Fanuc KAREL source: NC0061.KL

-- PROVISIONAL review KL for V940-1; original PC SHA256 46cbbacf586b5ee398f1359ac13f002e54e1b3793ebfd17aa1c9afa5b6356ba0
-- Incomplete behavior may be omitted. Consult companion uncertainty JSON. Do not deploy.
PROGRAM NC0061
%NOLOCKGROUP
-- UNRESOLVED_LOCAL_POOL 1 cells at code offset 3; source declarations unknown
-- DIRECT_LOCAL_WORD_ACCESS alone does not prove INTEGER, REAL, or BOOLEAN
BEGIN
  -- V9_CONDITION_STACK_HINT 10 bounded expression windows; static native code-base-relative target link; source arms held
  -- UNRESOLVED_PC offsets 0-8; opcodes 2B,2C,7B
  -- UNRESOLVED_PC offsets 13-20; opcodes 9D,23
  -- UNRESOLVED_PC offsets 25-42; opcodes 21,40,41,42
  -- UNRESOLVED_PC offsets 47-81; opcodes 21,2E,52,23,7A,40,41,42
  -- UNRESOLVED_PC offsets 86-110; opcodes 21,2E,52,23,7A,43
  -- UNRESOLVED_PC offsets 115-128; opcodes 21,9D,57,79
  -- UNRESOLVED_PC offsets 133-151; opcodes 21,2E,52,23
  -- UNRESOLVED_PC offsets 156-161; opcodes 7A
  -- UNRESOLVED_PC offsets 166-183; opcodes 21,40,41,42
  -- UNRESOLVED_PC offsets 188-222; opcodes 21,2E,52,23,7A,40,41,42
  -- UNRESOLVED_PC offsets 227-251; opcodes 21,2E,52,23,7A,43
  -- UNRESOLVED_PC offsets 256-269; opcodes 21,9D,57,79
  -- UNRESOLVED_PC offsets 274-292; opcodes 21,2E,52,23
  -- UNRESOLVED_PC offsets 297-302; opcodes 7A
  -- UNRESOLVED_PC offsets 307-324; opcodes 21,40,41,42
  -- UNRESOLVED_PC offsets 329-363; opcodes 21,2E,52,23,7A,40,41,42
  -- UNRESOLVED_PC offsets 368-392; opcodes 21,2E,52,23,7A,43
  -- UNRESOLVED_PC offsets 397-410; opcodes 21,9D,57,79
  -- UNRESOLVED_PC offsets 415-433; opcodes 21,2E,52,23
  -- UNRESOLVED_PC offsets 438-443; opcodes 7A
  -- UNRESOLVED_PC offsets 448-465; opcodes 21,40,41,42
  -- UNRESOLVED_PC offsets 470-504; opcodes 21,2E,52,23,7A,40,41,42
  -- UNRESOLVED_PC offsets 509-533; opcodes 21,2E,52,23,7A,43
  -- UNRESOLVED_PC offsets 538-551; opcodes 21,9D,57,79
  -- UNRESOLVED_PC offsets 556-574; opcodes 21,2E,52,23
  -- UNRESOLVED_PC offsets 579-584; opcodes 7A
  -- UNRESOLVED_PC offsets 589-606; opcodes 21,40,41,42
  -- UNRESOLVED_PC offsets 611-645; opcodes 21,2E,52,23,7A,40,41,42
  -- UNRESOLVED_PC offsets 650-674; opcodes 21,2E,52,23,7A,43
  -- UNRESOLVED_PC offsets 679-692; opcodes 21,9D,57,79
  -- UNRESOLVED_PC offsets 697-715; opcodes 21,2E,52,23
  -- UNRESOLVED_PC offsets 720-725; opcodes 7A
  -- UNRESOLVED_PC offsets 730-747; opcodes 21,40,41,42
  -- UNRESOLVED_PC offsets 752-786; opcodes 21,2E,52,23,7A,40,41,42
  -- UNRESOLVED_PC offsets 791-815; opcodes 21,2E,52,23,7A,43
  -- UNRESOLVED_PC offsets 820-833; opcodes 21,9D,57,79
  -- UNRESOLVED_PC offsets 838-856; opcodes 21,2E,52,23
  -- UNRESOLVED_PC offsets 861-866; opcodes 7A
  -- UNRESOLVED_PC offsets 871-888; opcodes 21,40,41,42
  -- UNRESOLVED_PC offsets 893-927; opcodes 21,2E,52,23,7A,40,41,42
  -- UNRESOLVED_PC offsets 932-956; opcodes 21,2E,52,23,7A,43
  -- UNRESOLVED_PC offsets 961-974; opcodes 21,9D,57,79
  -- UNRESOLVED_PC offsets 979-997; opcodes 21,2E,52,23
  -- UNRESOLVED_PC offsets 1002-1007; opcodes 7A
  -- UNRESOLVED_PC offsets 1012-1029; opcodes 21,40,41,42
  -- UNRESOLVED_PC offsets 1034-1068; opcodes 21,2E,52,23,7A,40,41,42
  -- UNRESOLVED_PC offsets 1073-1097; opcodes 21,2E,52,23,7A,43
  -- UNRESOLVED_PC offsets 1102-1115; opcodes 21,9D,57,79
  -- UNRESOLVED_PC offsets 1120-1138; opcodes 21,2E,52,23
  -- UNRESOLVED_PC offsets 1143-1148; opcodes 7A
  -- UNRESOLVED_PC offsets 1153-1170; opcodes 21,40,41,42
  -- UNRESOLVED_PC offsets 1175-1209; opcodes 21,2E,52,23,7A,40,41,42
  -- UNRESOLVED_PC offsets 1214-1238; opcodes 21,2E,52,23,7A,43
  -- UNRESOLVED_PC offsets 1243-1256; opcodes 21,9D,57,79
  -- UNRESOLVED_PC offsets 1261-1279; opcodes 21,2E,52,23
  -- UNRESOLVED_PC offsets 1284-1289; opcodes 7A
  -- UNRESOLVED_PC offsets 1294-1311; opcodes 21,40,41,42
  -- UNRESOLVED_PC offsets 1316-1350; opcodes 21,2E,52,23,7A,40,41,42
  -- UNRESOLVED_PC offsets 1355-1379; opcodes 21,2E,52,23,7A,43
  -- UNRESOLVED_PC offsets 1384-1397; opcodes 21,9D,57,79
  -- UNRESOLVED_PC offsets 1402-1420; opcodes 21,2E,52,23
  -- UNRESOLVED_PC offsets 1425-1430; opcodes 7A
  -- UNRESOLVED_PC offsets 1435-1449; opcodes 21,9D,52,23
  -- UNRESOLVED_PC offsets 1554-1558; opcodes 7F
  -- UNRESOLVED_PC offsets 1563-1567; opcodes 27,AA
  -- UNRESOLVED_PC offsets 1572-1576; opcodes 7F
END NC0061
